// TIA Portal V19 export
TYPE "UDT_STATUS_REQUEST"
   STRUCT
      in : Bool;
      acknIn : Bool;
      acknOut : Bool;
      out : "UDT_STATUS_SIM";
   END_STRUCT;
END_TYPE
